FUNCTION_BLOCK FB_HandScannerCtrl
VAR_INPUT
	bEnable				: BOOL;
	bReset				: BOOL;					(* set TRUE to clear RxBuffer and re-start COM line monitoring *)
	sFC1ReplacmentChar	: T_Char;
	bRemoveFNC1			: BOOL;
	sADSMasterNetID		: T_AmsNetId ;
	nSlaveAddr     	  		: UINT;
	eComPortMode		: ComSerialLineMode_t;	(* COM port type, PC/KL/EL COM ports can all be used *)
	nBaudRate			: UDINT;					(* data rate, e.g. 38400 = 38.4kbits/sec, max data rate depends on terminal type *)
	nDatabits			: BYTE;					(* no of databits for 1 character *)
	eParity				: ComParity_t;			(* PARITY_NONE, PARITY_EVEN or PARITY_ODD *)
	nStopbits			: BYTE;					(* no of stopbits *)
	tRXTimeOut			: TIME := T#350ms;
	nSizeComIn			: uINT;					(* size of ComIn buffer *)
	pComIn				: POINTER TO ARRAY[0..65] OF BYTE;	(* pointer to ComIn buffer *)
	pComOut				: POINTER TO ARRAY[0..65] OF BYTE;	(* pointer to ComOut buffer *)
	stHandScannerHostAck	:  ST_SCANNER_HostAck;
END_VAR
VAR_IN_OUT
	stHoneywellCtrl		:  ST_SCANNER_HoneywellCtrl;
END_VAR
VAR_OUTPUT

	bStringReceived			: BOOL;
	bExtStringReceived			: BOOL;
	bHandScanerPortOK			: BOOL;
	bHandScannerBaudrateOK	: BOOL;
	sScannerBarcode			: T_MaxString;
END_VAR
VAR

	fbHandScannerBaudrateMonitor 	: FB_SCANNER_BaudrateMonitor;
	bWrongBaudrateToWrite 			: BOOL;
	fbScannerCtrl					: FB_SCANNER_SerialCom_v2;
	sHandScannerTxBuffer			: ComBuffer;
	fbHandScannerCtrl				: FB_SCANNER_HoneyWellControl;

	tof_CheckComplete				: TOF;

END_VAR
VAR // added by the converter: edge detectors and wires of the graphical bodies
    _w1 : BOOL;
END_VAR

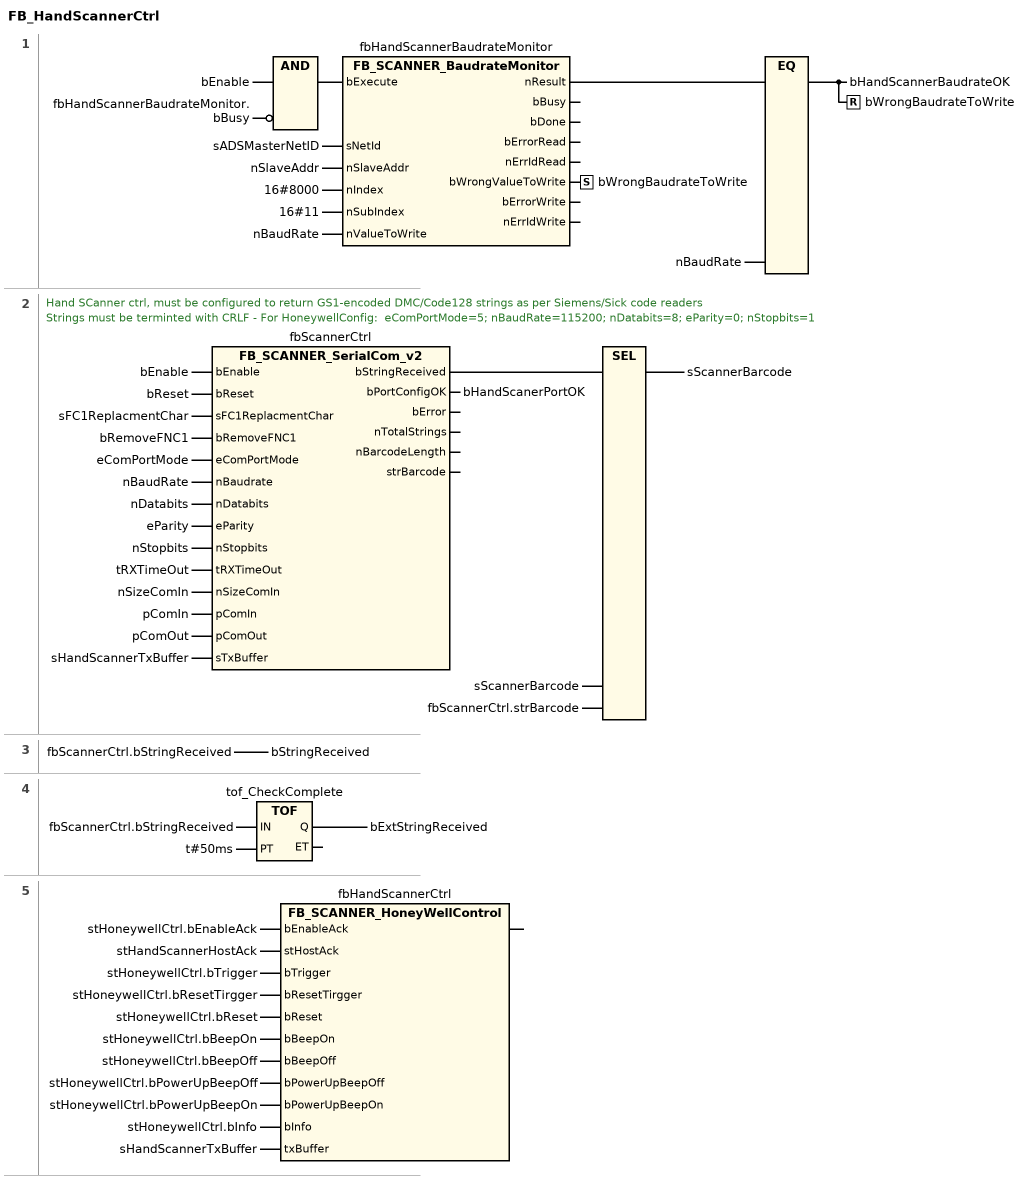
// NETWORK 1
fbHandScannerBaudrateMonitor(
    bExecute := bEnable AND NOT fbHandScannerBaudrateMonitor.bBusy,
    sNetId := sADSMasterNetID,
    nSlaveAddr := nSlaveAddr,
    nIndex := 16#8000,
    nSubIndex := 16#11,
    nValueToWrite := nBaudRate); // FB_SCANNER_BaudrateMonitor
bWrongBaudrateToWrite S= fbHandScannerBaudrateMonitor.bWrongValueToWrite;
_w1 := fbHandScannerBaudrateMonitor.nResult = nBaudRate;
bHandScannerBaudrateOK := _w1;
bWrongBaudrateToWrite R= _w1;

// NETWORK 2
// 					Hand SCanner ctrl, must be configured to return GS1-encoded DMC/Code128 strings as per Siemens/Sick code readers
// Strings must be terminted with CRLF - For HoneywellConfig:  eComPortMode=5; nBaudRate=115200; nDatabits=8; eParity=0; nStopbits=1
//
fbScannerCtrl(
    bEnable := bEnable,
    bReset := bReset,
    sFC1ReplacmentChar := sFC1ReplacmentChar,
    bRemoveFNC1 := bRemoveFNC1,
    eComPortMode := eComPortMode,
    nBaudrate := nBaudRate,
    nDatabits := nDatabits,
    eParity := eParity,
    nStopbits := nStopbits,
    tRXTimeOut := tRXTimeOut,
    nSizeComIn := nSizeComIn,
    pComIn := pComIn,
    pComOut := pComOut,
    sTxBuffer := sHandScannerTxBuffer,
    bPortConfigOK => bHandScanerPortOK); // FB_SCANNER_SerialCom_v2
sScannerBarcode := SEL(fbScannerCtrl.bStringReceived, sScannerBarcode, fbScannerCtrl.strBarcode);

// NETWORK 3
bStringReceived := fbScannerCtrl.bStringReceived;

// NETWORK 4
tof_CheckComplete(IN := fbScannerCtrl.bStringReceived, PT := t#50ms); // TOF
bExtStringReceived := tof_CheckComplete.Q;

// NETWORK 5
fbHandScannerCtrl(
    bEnableAck := stHoneywellCtrl.bEnableAck,
    stHostAck := stHandScannerHostAck,
    bTrigger := stHoneywellCtrl.bTrigger,
    bResetTirgger := stHoneywellCtrl.bResetTirgger,
    bReset := stHoneywellCtrl.bReset,
    bBeepOn := stHoneywellCtrl.bBeepOn,
    bBeepOff := stHoneywellCtrl.bBeepOff,
    bPowerUpBeepOff := stHoneywellCtrl.bPowerUpBeepOff,
    bPowerUpBeepOn := stHoneywellCtrl.bPowerUpBeepOn,
    bInfo := stHoneywellCtrl.bInfo,
    txBuffer := sHandScannerTxBuffer); // FB_SCANNER_HoneyWellControl

END_FUNCTION_BLOCK

(* stored: Version 1.1.0.1
   POU FB_HandScannerCtrl: Id {a44e3fd9-3acc-4003-8178-a38b3408d1f3}, SpecialFunc None *)
